Staubli VAL3: InstrItem.pjx

--- InstrItem.pjx ---
Parameters version=s7.2.1 stackSize=5000 millimeterUnit=true
Data file=InstrItem.dtx

--- InstrItem.dtx ---
public string sType
public string sData
